(* IEC 61131-3 sources: StewartPlatform/Class/DiasMasterPostScan, 1 file *)

(* ---- DiasMasterPostScan.st ---- *)
(*!
<Class
	Name               = "DiasMasterPostScan"
	Revision           = "1.0"
	RealtimeTask       = "false"
	CyclicTask         = "false"
	BackgroundTask     = "false"
	Sigmatek           = "true"
	OSInterface        = "false"
	HighPriority       = "true"
	Automatic          = "true"
	UpdateMode         = "Postscan"
	IconPath           = ".\Class\Tool.ico"
	SharedCommandTable = "true"
	Objectsize         = "(284,120)"
	Comment            = "to read inputs and to write the outputs in PostScan">
	<Channels>
		<Server Name="Server0" Visualized="false" Initialize="false" WriteProtected="true" Retentive="false"/>
		<Client Name="MasterConnect" Required="true" Internal="false" Comment="connection to Master "/>
	</Channels>
</Class>
*)
DiasMasterPostScan : CLASS
  //Servers:
	Server0 	: SvrChCmd_DINT;
  //Clients:
	MasterConnect 	: CltChCmd_DiasMaster;
  //Variables:
  //Functions:

	FUNCTION VIRTUAL GLOBAL CyWork
		VAR_INPUT
			EAX 	: UDINT := EAX;
		END_VAR
		VAR_OUTPUT
			state (EAX) 	: UDINT;
		END_VAR;
  //Tables:
	FUNCTION @STD
		VAR_OUTPUT
			ret_code	: CONFSTATES;
		END_VAR;
	FUNCTION GLOBAL TAB @CT_;
END_CLASS;

#pragma usingLtd DiasMaster

//*********************Inserted from .\DiasMasterPostScan\DiasMasterPostScan_00_00.st*********************

(****************************************************************************************
*
*	Created : Sigmatek
*	Changes :
*		0.0 => 1.0 / 23.12.2004 / no Mark / ws
*			compatibility with Lasal Class 2
*			removed visible flags from internal servers
*
*****************************************************************************************)
FUNCTION VIRTUAL GLOBAL DiasMasterPostScan::CyWork
VAR_INPUT
	EAX		: UDINT;
END_VAR
VAR_OUTPUT
	state		: UDINT;
END_VAR

	MasterConnect.CyWork(0);
	state:=READY;

END_FUNCTION //VIRTUAL GLOBAL DiasMasterPostScan::CyWork
